FUNCTION_BLOCK FB_ACL EXTENDS FB_CtrlBase
VAR
	// Specific interface struct for public access
	SIf: T_Ctrl_SIf_ACL;
	
	// Used blocks from lib. "utilities" for AMS route handling
	fbAddRoute:	FB_AddRouteEntry;
	
	// Used ADS blocks for communication
	fbWrite: ADSWRITE;
	fbRead: ADSREAD;
	fbReadWrite: ADSRDWRT;
		
	// List of all ADS connections handled by this block
	aListOfConnections: ARRAY[0..cuinMaxConnections] OF T_ADS_ConnectionData;
	
	// Number of ADS (server) connections
	uinNumOfAdsConnections: UINT;
	// Loop variable for request of the handle ID
	uinLoopReqHandle: UINT;
	// Connection index
	uinConIndex: UINT;	
	// Used for generate unique AMS route names
	uinRouteID: UINT;	
END_VAR
VAR CONSTANT
	// Sub states
	cSTA_SUB_INITIALIZE: INT := 500;
	cSTA_SUB_READ: INT := 501;
	cSTA_SUB_READBusy: INT := 502;
	cSTA_SUB_WRITE: INT := 503;
	cSTA_SUB_WRITEBusy: INT := 504;
	cSTA_SUB_RW: INT := 505;
	cSTA_SUB_RWBusy: INT := 506;
	cSTA_SUB_ADD_ROUTE: INT := 507;
	cSTA_SUB_ADD_ROUTEBusy: INT := 508;
	cSTA_SUB_ERROR: INT := 509;
	cSTA_SUB_DONE: INT := 510;
	cSTA_SUB_WAIT_NEXT_POLL: INT := 511;
END_VAR

(* Copyright 2017 Cimpress

Licensed under the Apache License, Version 2.0 (the "License");
you may not use this file except in compliance with the License.
You may obtain a copy of the License at

http://www.apache.org/licenses/LICENSE-2.0

Unless required by applicable law or agreed to in writing, software
distributed under the License is distributed on an "AS IS" BASIS,
WITHOUT WARRANTIES OR CONDITIONS OF ANY KIND, either express or implied.
See the License for the specific language governing permissions and
limitations under the License. *)

(*__________________________________________________________________________________________________
¦	
¦	Vistaprint Schweiz GmbH
¦	CH - 8401 Winterthur
¦
¦	www.vistaprint.ch - info@vistaprint.ch
¦___________________________________________________________________________________________________

Function desription:
ADS client for data exchange.
Controls the data exchange between various ADS devices. Devices can be added as server connections to that FUB. 

History:
Version		Date			Author		Comment
---------------------------------------------------------------------------------------------------
0.00.1		05.02.2014		AVME/DSC	Start history
0.00.2		17.02.2014		AVME/DSC	BugZilla 140 - Enter ADS route string automatically during state PONBusy

___________________________________________________________________________________________________*)

IF (me.bolActivate) THEN // cyclic call enabled
	IF (CIf.Info.bolInitDone=FALSE) THEN // first cycle -> init
		CtrlInit();
		CIf.Info.bolInitDone := TRUE;
	ELSE
		CycleStartDuty();
	
		Always();
		
		StateMachine();
		
		CycleEndDuty();
	
	END_IF
END_IF;

METHOD PROTECTED GetNextAccessType : INT
VAR_INPUT
	uinNextConnection:   UINT;
END_VAR
CASE aListOfConnections[uinNextConnection].eAccessType OF	
	E_ADS_AccessType.READ:
		GetNextAccessType:= cSTA_SUB_READ;	
	E_ADS_AccessType.WRITE:
		GetNextAccessType:= cSTA_SUB_WRITE;	
END_CASE
END_METHOD

METHOD PROTECTED sta_PONBusy : BOOL
VAR
	stRoute: ST_AmsRouteEntry;
	strRouteName: STRING;
END_VAR
// state implemetation
//--------------------------------------------------------------------------------------
// Entry action
	IF (me.StateMachine.intState<>me.StateMachine.intStateLastCycle) THEN
		me.StateMachine.intStateLastCycle := me.StateMachine.intState;
		
		uinRouteID:= 0;
		uinConIndex:=0;
		// Initialize sub state machine
		me.SubStateMachine.intState:= cSTA_SUB_ADD_ROUTE; 
		me.SubStateMachine.intStateNext := cSTA_SUB_ADD_ROUTE;
		
	END_IF

//--------------------------------------------------------------------------------------
// Cyclic action
	IF (me.StateMachine.intState=me.StateMachine.intStateLastCycle) THEN
		
			// Sub statemachine to set necessary AMS routes and determine the handle ID of all connections in list	
			CASE me.SubStateMachine.intState OF	
			
				// **************************************************************************
				// Call fbAddRoute to add AMS route. Block automatically check if NetID or Name already exist.
				// Double entries not possible!
				// **************************************************************************
				cSTA_SUB_ADD_ROUTE:
				
					// Prepare unique AMS route name: Controller Name: + ID
					uinRouteID:= uinRouteID + 1;
					strRouteName := CONCAT(CIf.Info.strName, ': ID');
					strRouteName := CONCAT(strRouteName, UINT_TO_STRING(uinRouteID));
							
					// Prepare route data
					stRoute.sName:= strRouteName;
					stRoute.sNetID:= aListOfConnections[uinConIndex].strNetID;
					stRoute.sAddress:= THIS^.NetIDtoAddress(aListOfConnections[uinConIndex].strNetID);
					stRoute.eTransport:= eRouteTransport_TCP_IP;
				
					// Add route
					fbAddRoute(bExecute	:= FALSE);
					fbAddRoute( sNetID 	:= '',
								stRoute	:= stRoute,
								bExecute:= TRUE,
								tTimeout:= UDINT_TO_TIME(SIf.Par.udiTOAddRoute_ms),
								bBusy	=>,
								bError	=>,
								nErrID	=>);
				
					me.SubStateMachine.intStateNext := cSTA_SUB_ADD_ROUTEBusy;		
							
				// **************************************************************************
				// Add route busy
				// **************************************************************************
				cSTA_SUB_ADD_ROUTEBusy:
				
					fbAddRoute(bExecute:= FALSE);
					// Add route done
					IF NOT (fbAddRoute.bBusy) THEN
						IF NOT (fbAddRoute.bError) THEN
							// More connections?
							IF (uinConIndex < (uinNumOfAdsConnections-1)) THEN
								uinConIndex:= uinConIndex+1;
								me.SubStateMachine.intStateNext := cSTA_SUB_ADD_ROUTE;
							// All routes added - go on with determine the handle ID 
							ELSE
								uinConIndex:=0;
								me.SubStateMachine.intStateNext := cSTA_SUB_RW;	
							END_IF
						// Error
						ELSE
							// SIf.Alm[7].strText :=  'Adding AMS route failed. Note add. info for affected connection ID';
							pfbAlarmCtrl^.setAlarm(CIf.Info.intCtrlId,7,UDINT_TO_DINT(aListOfConnections[uinConIndex].udiConID),ADR(SIf.Alm),E_AlmState.RST,CIf.Job.eMe_ActivAlmClass);
							me.SubStateMachine.intStateNext := cSTA_SUB_ERROR;		
						END_IF
					END_IF
			
				// **************************************************************************
				// Call fbReadWrite to determine the handle ID
				// **************************************************************************
				cSTA_SUB_RW:
			
					fbReadWrite(WRTRD:= FALSE);
    				fbReadWrite(NETID		:= aListOfConnections[uinConIndex].strNetID,
                				PORT		:= aListOfConnections[uinConIndex].uinTargetPort,
                   				IDXGRP		:= cGET_SYMHANDLE_BYNAME,  
                   				IDXOFFS     := 16#0000,
                   				WRITELEN    := INT_TO_UDINT(LEN(aListOfConnections[uinConIndex].strRoute)+1),
								READLEN     := SIZEOF(aListOfConnections[uinConIndex].udiHandle),
								SRCADDR     := ADR(aListOfConnections[uinConIndex].strRoute),
								DESTADDR    := ADR(aListOfConnections[uinConIndex].udiHandle),
								WRTRD       := TRUE,
								TMOUT       := UDINT_TO_TIME(SIf.Par.udiTORWData_ms),
								BUSY        => ,
								ERR         => ,
								ERRID       => );
								
					me.SubStateMachine.intStateNext := cSTA_SUB_RWBusy;		
				
				// **************************************************************************
				// Read/Write busy
				// **************************************************************************
				cSTA_SUB_RWBusy:
					fbReadWrite(WRTRD:= FALSE);
					// Read/Write done
					IF NOT (fbReadWrite.BUSY) THEN
						IF NOT (fbReadWrite.ERR) THEN
							// More connections?
							IF (uinConIndex < (uinNumOfAdsConnections-1)) THEN
								uinConIndex:= uinConIndex+1;
								me.SubStateMachine.intStateNext := cSTA_SUB_RW;
							// Done - all connection handles are determined 
							ELSE
								me.SubStateMachine.intStateNext := cSTA_SUB_DONE;	
							END_IF
						// Error
						ELSE
							// SIf.Alm[3].strText := 'Init of ADS connection failed. Check add. info for affected connection ID';
							pfbAlarmCtrl^.setAlarm(CIf.Info.intCtrlId,3,UDINT_TO_DINT(aListOfConnections[uinConIndex].udiConID),ADR(SIf.Alm),E_AlmState.RST,CIf.Job.eMe_ActivAlmClass);
							me.SubStateMachine.intStateNext := cSTA_SUB_ERROR;		
						END_IF
					END_IF
				
				// **************************************************************************
				// All necessary AMS routes set and connection handles are determined 
				// **************************************************************************
				cSTA_SUB_DONE:
				
				// **************************************************************************
				// Error
				// **************************************************************************
				cSTA_SUB_ERROR:
				
			END_CASE	
			
		
		// State Change Condition
		IF ((me.SubStateMachine.intState=cSTA_SUB_ERROR) OR (me.StateMachine.udiTimeInState_ms >= SIf.Par.udiTOPowerOn_ms)) THEN
			// In case if TO
			IF (me.StateMachine.udiTimeInState_ms >= SIf.Par.udiTOPowerOn_ms) THEN
				// SIf.Alm[2].strText := 'Timeout initialize ADS connection(s)';
				pfbAlarmCtrl^.setAlarm(CIf.Info.intCtrlId,2,UDINT_TO_DINT(me.StateMachine.udiTimeInState_ms),ADR(SIf.Alm),E_AlmState.RST,CIf.Job.eMe_ActivAlmClass);
			END_IF
			me.StateMachine.intStateNext := cSTA_ERROR;				
		ELSIF (me.SubStateMachine.intState=cSTA_SUB_DONE) THEN
			me.StateMachine.intStateNext := cSTA_PON;
		END_IF
			
	END_IF

//--------------------------------------------------------------------------------------
// Exit action
	IF (me.StateMachine.intState<>me.StateMachine.intStateNext) THEN
		;
	END_IF
END_METHOD

METHOD PROTECTED sta_RUNBusy : BOOL
// state implemetation
//--------------------------------------------------------------------------------------
// Entry action
	IF (me.StateMachine.intState<>me.StateMachine.intStateLastCycle) THEN
		me.StateMachine.intStateLastCycle := me.StateMachine.intState;
		;
	END_IF

//--------------------------------------------------------------------------------------
// Cyclic action
	IF (me.StateMachine.intState=me.StateMachine.intStateLastCycle) THEN
		IF (TRUE) THEN
			me.StateMachine.intStateNext := BASE_PLC.cSTA_RUN;
		END_IF
	END_IF

//--------------------------------------------------------------------------------------
// Exit action
	IF (me.StateMachine.intState<>me.StateMachine.intStateNext) THEN
		;
	END_IF
END_METHOD

METHOD PROTECTED sta_RUN : BOOL
// state implemetation
//--------------------------------------------------------------------------------------
// Entry action
	IF (me.StateMachine.intState<>me.StateMachine.intStateLastCycle) THEN
		me.StateMachine.intStateLastCycle := me.StateMachine.intState;
					
		uinConIndex:=0;
		// Initialize sub state machine
		me.SubStateMachine.intState:= cSTA_SUB_INITIALIZE; 
		me.SubStateMachine.intStateNext := cSTA_SUB_INITIALIZE;
	END_IF

//--------------------------------------------------------------------------------------
// Cyclic action
	IF (me.StateMachine.intState=me.StateMachine.intStateLastCycle) THEN

		// Sub statemachine to handle all connections in list dependent access type (read, write, rw)
		CASE me.SubStateMachine.intState OF	
	
			//************************************************************************
			// Initialize
			//************************************************************************
			cSTA_SUB_INITIALIZE:
				// Get access type
				me.SubStateMachine.intStateNext:= THIS^.GetNextAccessType(uinConIndex);
							
			//************************************************************************					
			// Call fbRead
			//************************************************************************
			cSTA_SUB_READ:
		
				fbRead(READ:= FALSE);
				fbRead(NETID       := aListOfConnections[uinConIndex].strNetID,
						PORT       := aListOfConnections[uinConIndex].uinTargetPort,
						IDXGRP     := cREAD_WRITE_SYMVAL_BYHANDLE,
						IDXOFFS    := aListOfConnections[uinConIndex].udiHandle,
						LEN        := aListOfConnections[uinConIndex].udiDataLen,
						DESTADDR   := aListOfConnections[uinConIndex].pData,
						READ       := TRUE,
						TMOUT      := UDINT_TO_TIME(SIf.Par.udiTOReadData_ms),
						BUSY       => ,
						ERR        => ,
						ERRID      => );
														
				me.SubStateMachine.intStateNext := cSTA_SUB_READBusy;			
							
			//************************************************************************
			// Read busy
			//************************************************************************
			cSTA_SUB_READBusy:
				fbRead(READ:= FALSE);
				// Read done
				IF NOT (fbRead.BUSY) THEN
					IF NOT (fbRead.ERR) THEN	
						// More connections?
						IF (uinConIndex < (uinNumOfAdsConnections-1)) THEN
							uinConIndex:= uinConIndex+1;
							// Get next access type
							me.SubStateMachine.intStateNext:= THIS^.GetNextAccessType(uinConIndex);
						// Done - all connection handles are determined 
						ELSE
							me.SubStateMachine.intStateNext := cSTA_SUB_WAIT_NEXT_POLL;	
						END_IF						
					// Error
					ELSE
						// SIf.Alm[4].strText := 'ADS read data failed. Note add. info to get ADS error ID';
						pfbAlarmCtrl^.setAlarm(CIf.Info.intCtrlId,4,UDINT_TO_DINT(fbRead.ERRID),ADR(SIf.Alm),E_AlmState.RST,CIf.Job.eMe_ActivAlmClass);
						me.SubStateMachine.intStateNext := cSTA_SUB_ERROR;		
					END_IF
				END_IF	
				
			//************************************************************************					
			// Call fbWrite
			//************************************************************************
			cSTA_SUB_WRITE:
		
				fbWrite(WRITE:= FALSE);
				fbWrite(NETID      := aListOfConnections[uinConIndex].strNetID,
						PORT       := aListOfConnections[uinConIndex].uinTargetPort,
						IDXGRP     := cREAD_WRITE_SYMVAL_BYHANDLE,
						IDXOFFS    := aListOfConnections[uinConIndex].udiHandle,
						LEN        := aListOfConnections[uinConIndex].udiDataLen,
						SRCADDR    := aListOfConnections[uinConIndex].pData,
						WRITE      := TRUE,
						TMOUT      := UDINT_TO_TIME(SIf.Par.udiTOWriteData_ms),
						BUSY       => ,
						ERR        => ,
						ERRID      => );
														
				me.SubStateMachine.intStateNext := cSTA_SUB_WRITEBusy;		
				
			//************************************************************************
			// Write busy
			//************************************************************************
			cSTA_SUB_WRITEBusy:
				fbWrite(WRITE:= FALSE);
				// Write done
				IF NOT (fbWrite.BUSY) THEN
					IF NOT (fbWrite.ERR) THEN
						// More connections?
						IF (uinConIndex < (uinNumOfAdsConnections-1)) THEN
							uinConIndex:= uinConIndex+1;
							// Get next access type
							me.SubStateMachine.intStateNext:= THIS^.GetNextAccessType(uinConIndex);
						// Done - all connection handles are determined 
						ELSE
							me.SubStateMachine.intStateNext := cSTA_SUB_WAIT_NEXT_POLL;	
						END_IF
					// Error
					ELSE
						// SIf.Alm[5].strText := 'ADS write data failed. Note add. info to get ADS error ID';
						pfbAlarmCtrl^.setAlarm(CIf.Info.intCtrlId,5,UDINT_TO_DINT(fbWrite.ERRID),ADR(SIf.Alm),E_AlmState.RST,CIf.Job.eMe_ActivAlmClass);
						me.SubStateMachine.intStateNext := cSTA_SUB_ERROR;		
					END_IF
				END_IF			
		
			//************************************************************************
			// Wait for next polling - Connection list completely processed 
			//************************************************************************	
			cSTA_SUB_WAIT_NEXT_POLL:
			
				// Wait polling time expired 	
				IF (me.SubStateMachine.udiTimeInState_ms >= SIf.Par.udiPollingInterval_ms) THEN				
					//Start again at first connection in list
					uinConIndex:=0;
					me.SubStateMachine.intStateNext := cSTA_SUB_INITIALIZE;
				END_IF
				
			//************************************************************************
			// ERROR			
			//************************************************************************	
			cSTA_SUB_ERROR:
				// SIf.Alm[6].strText := 'ADS connection fault. Note add. info for affected connection ID';
				pfbAlarmCtrl^.setAlarm(CIf.Info.intCtrlId,6,UDINT_TO_DINT(aListOfConnections[uinConIndex].udiConID),ADR(SIf.Alm),E_AlmState.RST,CIf.Job.eMe_ActivAlmClass);
				me.StateMachine.intStateNext := BASE_PLC.cSTA_ERROR;	
			
		END_CASE			
	END_IF

//--------------------------------------------------------------------------------------
// Exit action
	IF (me.StateMachine.intState<>me.StateMachine.intStateNext) THEN
		;
	END_IF
END_METHOD

METHOD AddConnection
VAR_INPUT
	stConnection: T_ADS_ConnectionData;
END_VAR
// Method adds a connection to the internal list of all ADS connections handled by this block
IF (uinNumOfAdsConnections <= (cuinMaxConnections-1)) THEN
	// Add connection to list
	aListOfConnections[uinNumOfAdsConnections] := stConnection;
	// Assigned connection ID
	aListOfConnections[uinNumOfAdsConnections].udiConID := uinNumOfAdsConnections+1;
	// Inc. number of connections
	uinNumOfAdsConnections:= uinNumOfAdsConnections+1;
END_IF
END_METHOD

PROPERTY PUBLIC CtrlSIf : POINTER TO T_Ctrl_SIf_ACL
GET
CtrlSIf := ADR(SIf);
END_GET
END_PROPERTY

METHOD PROTECTED StateMachine : BOOL
SUPER^.StateMachine();

// main statemachine of base controller
CASE me.StateMachine.intState OF
	cSTA_RUNBusy: 
        THIS^.sta_RUNBusy();
    cSTA_RUN: 
        THIS^.sta_RUN();				
END_CASE;
END_METHOD

METHOD PROTECTED getCmdState : STRING
VAR_INPUT
	intCmdState: INT;
	bolState: BOOL;
END_VAR
getCmdState := SUPER^.getCmdState(intCmdState:=intCmdState,bolState:=bolState); // get global/base defined cmds/states
IF (getCmdState='') THEN // global not defined get local
	// get string cmd/state string information in runtime
	IF (bolState=FALSE) THEN
		(*
		// cmd's
		CASE intCmdState OF
			;
		END_CASE
		*)
	ELSE
		// states
		CASE intCmdState OF
			// SUB States
			cSTA_SUB_INITIALIZE:
				getCmdState := 'cSTA_SUB_INITIALIZE';
			cSTA_SUB_READ:
				getCmdState := 'cSTA_SUB_READ';
			cSTA_SUB_READBusy:
				getCmdState := 'cSTA_SUB_READBusy';
			cSTA_SUB_WRITE:
				getCmdState := 'cSTA_SUB_WRITE';
			cSTA_SUB_WRITEBusy:
				getCmdState := 'cSTA_SUB_WRITEBusy';			
			cSTA_SUB_RW:
				getCmdState := 'cSTA_SUB_RW';
			cSTA_SUB_RWBusy:
				getCmdState := 'cSTA_SUB_RWBusy';	
			cSTA_SUB_ADD_ROUTE:
				getCmdState := 'cSTA_SUB_ADD_ROUTE';	
			cSTA_SUB_ADD_ROUTEBusy:
				getCmdState := 'cSTA_SUB_ADD_ROUTEBusy';			
			cSTA_SUB_ERROR:
				getCmdState := 'cSTA_SUB_ERROR';
			cSTA_SUB_DONE:
				getCmdState := 'cSTA_SUB_DONE';
			cSTA_SUB_WAIT_NEXT_POLL:
				getCmdState := 'cSTA_SUB_WAIT_NEXT_POLL';
		END_CASE
	END_IF
END_IF
END_METHOD

METHOD getCtrlSIf : POINTER TO T_Ctrl_SIf_ACL
getCtrlSIf := ADR(SIf);
END_METHOD

METHOD PROTECTED sta_OFF : BOOL
// state implemetation
//--------------------------------------------------------------------------------------
// Entry action
	IF (me.StateMachine.intState<>me.StateMachine.intStateLastCycle) THEN
		me.StateMachine.intStateLastCycle := me.StateMachine.intState;
		// Initialize sub state machine
		me.SubStateMachine.intState:= cSTA_SUB_INITIALIZE; 
		me.SubStateMachine.intStateNext := cSTA_SUB_INITIALIZE;
	END_IF
	
//--------------------------------------------------------------------------------------
// Cyclic action
	IF (me.StateMachine.intState=me.StateMachine.intStateLastCycle) THEN	
		// State Change Condition
		IF (me.Alarm.eActivAlmClass<>E_AlmClass.EOFF) AND (me.Alarm.eActivAlmClass<>E_AlmClass.OFF) THEN	
			IF(me.intCmd=BASE_PLC.cCMD_RUN) THEN
				me.StateMachine.intStateNext := BASE_PLC.cSTA_RUNBusy;
			END_IF
		END_IF
	END_IF

//--------------------------------------------------------------------------------------
// Exit action
	IF (me.StateMachine.intState<>me.StateMachine.intStateNext) THEN
		;
	END_IF
END_METHOD

METHOD PROTECTED Always : BOOL
SUPER^.Always();

// ----------------------------------------------------------------------------------
// cyclic actions outside of statemachine
IF (me.StateMachine.intState<>cSTA_SINGLE_ANSWER) THEN
	SIf.Cur.uinNumOfAdsConnections:= uinNumOfAdsConnections;	
END_IF

// If no connection added, set alarm and change to state error
IF (uinNumOfAdsConnections = 0) THEN
	// Set Alarm: SIf.Alm[1].strText := 'Initialization error. Minimum one ADS connection must be configured'; 
	pfbAlarmCtrl^.setAlarm(CIf.Info.intCtrlId,1,0,ADR(SIf.Alm),E_AlmState.RST,CIf.Job.eMe_ActivAlmClass);	
	me.StateMachine.intStateNext := BASE_PLC.cSTA_ERROR;
END_IF

// ----------------------------------------------------------------------------------
// Always change actions in Base Library
// ----------------------------------------------------------------------------------
// overrule error always from base -> no EOFF State!! in EOFF go to OFF
IF (me.StateMachine.intStateNext = cSTA_EOFFBusy) THEN
	IF (me.StateMachine.intState=cSTA_OFF) THEN
		me.StateMachine.intStateNext := cSTA_OFF;
	ELSE // stay in OFF
		me.StateMachine.intStateNext := cSTA_OFFBusy;
	END_IF
END_IF
END_METHOD

METHOD PROTECTED sta_PON : BOOL
// state implemetation
//--------------------------------------------------------------------------------------
// Entry action
	IF (me.StateMachine.intState<>me.StateMachine.intStateLastCycle) THEN
		me.StateMachine.intStateLastCycle := me.StateMachine.intState;
		
	END_IF

//--------------------------------------------------------------------------------------
// Cyclic action
	IF (me.StateMachine.intState=me.StateMachine.intStateLastCycle) THEN
		
		;	
		// State Change Condition
		IF (me.intCmd<>cCMD_PON) AND (me.intCmd<>cCMD_DONE) THEN
			me.StateMachine.intStateNext := BASE_PLC.cSTA_OFFBusy;
		END_IF
	END_IF

//--------------------------------------------------------------------------------------
// Exit action
	IF (me.StateMachine.intState<>me.StateMachine.intStateNext) THEN
		;
	END_IF
END_METHOD

METHOD NetIDtoAddress: STRING
VAR_INPUT
	strNetID: STRING;
END_VAR
VAR
	intI: INT;
	strCharacter: STRING(1);
	uinExitCounter: UINT;
	cDot: USINT := 16#2E;
END_VAR
// Method convert a ADS NetID to a standard IP Address
// Example: 192.168.70.27.1.1 -> 192.168.70.27
uinExitCounter:=0;
// Get all numbers up to 4 point
FOR intI:=0 TO LEN(strNetID) DO	
	// Get single char
	strCharacter:= Mid(strNetID,1,intI);
	// Incr. exit counter if char = '.'
	IF (F_ToASC(strCharacter) = cDot) THEN
		uinExitCounter:= uinExitCounter +1;
	END_IF
	// As long as 4 point not reached
	IF uinExitCounter < 4 THEN
		NetIDtoAddress:= CONCAT(NetIDtoAddress,strCharacter);	
	ELSE
		EXIT;
	END_IF 
END_FOR
END_METHOD

METHOD FB_init : BOOL
VAR_INPUT
	///if TRUE, the retain variables are initialized (warm start / cold start)
	bInitRetains: BOOL;
	///if TRUE, the instance afterwards gets moved into the copy code (online change)
	bInCopyCode: BOOL;
END_VAR
VAR
	udiTaskCnt: UDINT;
	ii: UINT;
END_VAR
//------------------------------------------------------------------------------------------------------------------------
// to manually change in new FUB implementation!!!
// define valid commands for this controller
FOR ii:= 0 TO (SIZEOF(CIf.Job.aCmdList)/SIZEOF(CIf.Job.aCmdList[0])-1) BY 1 DO
	IF (CIf.Job.aCmdList[ii].intCmd=cCMD_INITIALIZED) THEN
		// found first empty array element
		EXIT;
	END_IF
END_FOR
CIf.Job.aCmdList[ii].intCmd := cCMD_RUN;
CIf.Job.aCmdList[ii].strName := 'Run'; 
CIf.Job.aCmdList[ii].bolAvailable := TRUE;
ii := ii +1;

// set name of class/typ
CIf.Info.strType := 'FB_ACL';
CIf.Info.strFullName := 'ADS Client';

// set alarm class
SIf.Alm[1].eAlmClass := E_AlmClass.OFF;
SIf.Alm[1].strText := 'Initialization error. Minimum one ADS connection must be configured'; 
SIf.Alm[2].eAlmClass := E_AlmClass.OFF;
SIf.Alm[2].strText := 'Timeout initialize ADS connection(s)';
SIf.Alm[3].eAlmClass := E_AlmClass.OFF;
SIf.Alm[3].strText := 'Init of ADS connection failed. Note add. info for affected connection ID';
SIf.Alm[4].eAlmClass := E_AlmClass.OFF;
SIf.Alm[4].strText := 'ADS read data failed. Note add. info to get ADS error ID';
SIf.Alm[5].eAlmClass := E_AlmClass.OFF;
SIf.Alm[5].strText := 'ADS write data failed. Note add. info to get ADS error ID';
SIf.Alm[6].eAlmClass := E_AlmClass.OFF;
SIf.Alm[6].strText := 'ADS connection fault. Note add. info for affected connection ID';
SIf.Alm[7].eAlmClass := E_AlmClass.OFF;
SIf.Alm[7].strText :=  'Adding AMS route failed. Note add. info for affected connection ID';

//*******************************************************************************
// initial values
//*******************************************************************************

// software configuration
CIf.SwCfg.bolExist := TRUE;
CIf.SwCfg.bolSimulation := FALSE;

// parameter
SIf.Par.udiTOAddRoute_ms:= 1500;
SIf.Par.udiTOPowerOn_ms:= 10000;
SIf.Par.udiTOReadData_ms:= 1500;
SIf.Par.udiTOWriteData_ms:= 1500;
SIf.Par.udiTORWData_ms:= 1500;
SIf.Par.udiPollingInterval_ms:= 100;
END_METHOD

METHOD PROTECTED sta_ERROR : BOOL
// state implemetation
//--------------------------------------------------------------------------------------
// Entry action
	IF (me.StateMachine.intState<>me.StateMachine.intStateLastCycle) THEN
		me.StateMachine.intStateHistory := me.StateMachine.intStateLastCycle; // -> possibillity to go back to state before error
		me.StateMachine.intStateLastCycle := me.StateMachine.intState;
		
		// Initialize sub state machine
		me.SubStateMachine.intState:= cSTA_SUB_INITIALIZE; 
		me.SubStateMachine.intStateNext := cSTA_SUB_INITIALIZE;
	END_IF

//--------------------------------------------------------------------------------------
// Cyclic action
	IF (me.StateMachine.intState=me.StateMachine.intStateLastCycle) THEN
		// State Change Condition
		IF (CIf.Job.bolAlmReset = TRUE) THEN
			me.StateMachine.intStateNext := cSTA_ERRORQuit;
		END_IF
	END_IF

//--------------------------------------------------------------------------------------
// Exit action
	IF (me.StateMachine.intState<>me.StateMachine.intStateNext) THEN
		;
	END_IF
END_METHOD

END_FUNCTION_BLOCK

(* stored: Version 1.1.0.1, ProductVersion 3.1.4019.2
   POU FB_ACL: Id {35c44579-8ee6-4bc6-a332-f87fe74b8d5d}, SpecialFunc None
   Method GetNextAccessType: Id {096217a9-b3f5-4913-8799-35029a3ae704}
   Method sta_PONBusy: Id {10205a02-c205-4a68-aa3f-517c69831d55}
   Method sta_RUNBusy: Id {17796103-9d26-4e6c-8d4b-5a11d68fbae7}
   Method sta_RUN: Id {1eadda75-9ac1-47cb-b64c-ca5613f16207}
   Method AddConnection: Id {2e3aa29c-2c8b-4b4e-b83b-bda7f50bd268}
   Property CtrlSIf: Id {309b1a1d-faae-42bc-9507-42d211c6d40e}
   Get Get: Id {155f0f78-526f-462c-891a-0145f6676d2f}
   Method StateMachine: Id {3c973f2a-7cfa-4400-8508-f52d5e67adff}
   Method getCmdState: Id {48c1ab59-ea2d-486d-bdfb-c97920a611f0}
   Method getCtrlSIf: Id {5bcded1c-e34b-4dd0-82f9-810996aa589a}
   Method sta_OFF: Id {82e22428-a03a-4e02-9fcd-a314f0399cc9}
   Method Always: Id {83199abc-a2c6-42b3-97c5-faf95e44d62f}
   Method sta_PON: Id {bae7231a-f1c3-4551-a7da-0fd79e4b7301}
   Method NetIDtoAddress: Id {d12b7a94-c50c-4873-88a2-9a106eb6cd59}
   Method FB_init: Id {da026435-4584-4f7d-b3e7-ef72bcf894b2}
   Method sta_ERROR: Id {f00aa3c1-1388-4d00-961e-356b78c04a4b} *)
